TYPE ST_Com_ExportStation :
STRUCT
		IN: 		ST_ComIn_ExportStation;
		OUT:		ST_ComOut_ExportStation;
		ManualMovement: ST_ManMov_Station;
END_STRUCT
END_TYPE

(* stored: Version 1.1.0.1
   DUT ST_Com_ExportStation: Id {b1b6a454-2fc5-47e7-abd5-9914d947d331} *)
